// TIA Portal V17 export
// export: Created 2024-09-03T21:54:47.1787587Z, ExportSetting WithDefaults, DisplayName Totally Integrated Automation Portal, DisplayVersion V17 Update 7, DisplayName TIA Portal Openness, DisplayVersion V17 Update 7, DisplayName TIA Portal Version Control Interface, DisplayVersion V17, DisplayName SINAMICS Startdrive Advanced, DisplayVersion V17 SP2, DisplayName SINAMICS Startdrive G110M, G120, G120C, G120D, G120P, G115D, DisplayVersion V17 SP2, DisplayName SINAMICS Startdrive G130, G150, S120, S150, SINAMICS MV, S210, DisplayVersion V17 SP2, DisplayName STEP 7 Professional, DisplayVersion V17 Update 7, DisplayName STEP 7 Safety, DisplayVersion V17 Update 6, DisplayName WinCC Advanced / Unified PC, DisplayVersion V17 Update 7
FUNCTION "FC_BitsToUInt" : Void   // FC1020, LAD
{ S7_Optimized_Access := 'FALSE' }
VERSION : 0.1
// stored: AutoNumber false, IsIECCheckEnabled false, SetENOAutomatically false, UDAEnableTagReadback false
   VAR_INPUT
      iBit1 : Bool;
      iBit2 : Bool;
      iBit3 : Bool;
      iBit4 : Bool;
      iBit5 : Bool;
      iBit6 : Bool;
      iBit7 : Bool;
      iBit8 : Bool;
      iBit9 : Bool;
      iBit10 : Bool;
      iBit11 : Bool;
      iBit12 : Bool;
      iBit13 : Bool;
      iBit14 : Bool;
      iBit15 : Bool;
      iBit16 : Bool;
   END_VAR
   VAR_OUTPUT
      qValue : UInt;
   END_VAR
   VAR_TEMP
      value : UInt;
   END_VAR
BEGIN

REGION Network 1: Convert bits to UInt
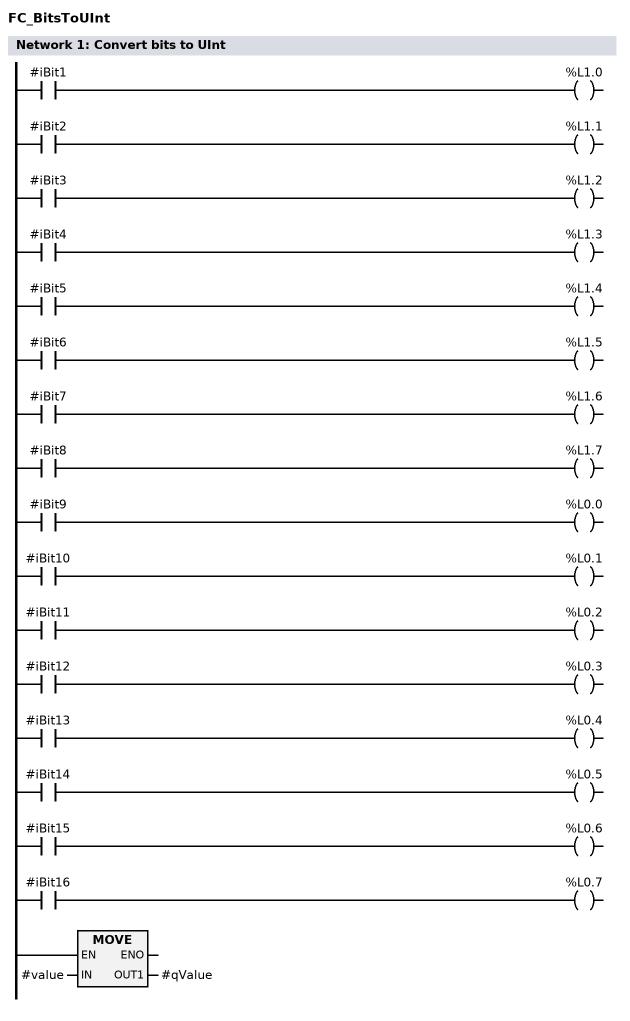
   RUNG wire#powerrail
      Contact( #iBit1 )
      Coil( %L1.0 )
   END_RUNG
   RUNG wire#powerrail
      Contact( #iBit2 )
      Coil( %L1.1 )
   END_RUNG
   RUNG wire#powerrail
      Contact( #iBit3 )
      Coil( %L1.2 )
   END_RUNG
   RUNG wire#powerrail
      Contact( #iBit4 )
      Coil( %L1.3 )
   END_RUNG
   RUNG wire#powerrail
      Contact( #iBit5 )
      Coil( %L1.4 )
   END_RUNG
   RUNG wire#powerrail
      Contact( #iBit6 )
      Coil( %L1.5 )
   END_RUNG
   RUNG wire#powerrail
      Contact( #iBit7 )
      Coil( %L1.6 )
   END_RUNG
   RUNG wire#powerrail
      Contact( #iBit8 )
      Coil( %L1.7 )
   END_RUNG
   RUNG wire#powerrail
      Contact( #iBit9 )
      Coil( %L0.0 )
   END_RUNG
   RUNG wire#powerrail
      Contact( #iBit10 )
      Coil( %L0.1 )
   END_RUNG
   RUNG wire#powerrail
      Contact( #iBit11 )
      Coil( %L0.2 )
   END_RUNG
   RUNG wire#powerrail
      Contact( #iBit12 )
      Coil( %L0.3 )
   END_RUNG
   RUNG wire#powerrail
      Contact( #iBit13 )
      Coil( %L0.4 )
   END_RUNG
   RUNG wire#powerrail
      Contact( #iBit14 )
      Coil( %L0.5 )
   END_RUNG
   RUNG wire#powerrail
      Contact( #iBit15 )
      Coil( %L0.6 )
   END_RUNG
   RUNG wire#powerrail
      Contact( #iBit16 )
      Coil( %L0.7 )
   END_RUNG
   RUNG wire#powerrail
      Move(in := #value, out1 => #qValue)
   END_RUNG
   // the same network as SCL:
   %L1.0 := #iBit1;
   %L1.1 := #iBit2;
   %L1.2 := #iBit3;
   %L1.3 := #iBit4;
   %L1.4 := #iBit5;
   %L1.5 := #iBit6;
   %L1.6 := #iBit7;
   %L1.7 := #iBit8;
   %L0.0 := #iBit9;
   %L0.1 := #iBit10;
   %L0.2 := #iBit11;
   %L0.3 := #iBit12;
   %L0.4 := #iBit13;
   %L0.5 := #iBit14;
   %L0.6 := #iBit15;
   %L0.7 := #iBit16;
   #qValue := #value;
END_REGION
END_FUNCTION
